# EPICS substitutions: asubtestApp/Db/modifyevrseq.substitutions
file evrcalcdelay.template
{
pattern {SYS, DEV}
	{$(SYS), $(DEV1)}
	{$(SYS), $(DEV2)}
	{$(SYS), $(DEV3)}
	{$(SYS), $(DEV4)}
}

file asubseq.template
{
pattern {SYS, EVR}
	{$(SYS), $(EVR)}
}
